{attribute 'qualified_only'}
{attribute 'strict'}
{attribute 'to_string'}
TYPE E_PROCESS_CHECK :
(
  NULL,
  REFERENCE_CTRL_INVALID,
  REFERENCE_STATE_INVALID,
  REFERENCE_MOVER_INFO_INVALID,
	STATION_FIRST_ZERO,
  STATION_LAST_ZERO,
  STATION_FIRST_MAX,
  STATION_LAST_MAX,
  STATION_COUNT_NEGATIVE, // last station must have higher index than first station, range must also be closed
  STATION_COUNT_TOO_HIGH, // process can only be max (SIZEOF(T_PROCESS)*8)

  CHECK_DONE    := 10000
);
END_TYPE

(* stored: Version 1.1.0.1, ProductVersion 3.1.4026.18
   DUT E_PROCESS_CHECK: Id {13181fdf-4b05-48d0-980c-6977717334ca} *)
